// TIA Portal V16 export
// export: Created 2024-12-03T15:41:46.0079114Z, ExportSetting WithReadOnly, DisplayName Totally Integrated Automation Portal, DisplayVersion V16 Update 6, DisplayName TIA Portal Version Control Interface, DisplayVersion V16 Update 2, DisplayName TIA Portal Openness, DisplayVersion V16 Update 6, DisplayName TIA Portal Teamcenter Gateway, DisplayVersion V16, DisplayName SINAMICS Startdrive Advanced, DisplayVersion V16 Update 5, DisplayName SINAMICS Startdrive G130, G150, S120, S150, SINAMICS MV, S210, DisplayVersion V16 Update 5, DisplayName SINAMICS Startdrive G110M, G120, G120C, G120D, G120P, G115D, DisplayVersion V16 Update 5, DisplayName STEP 7 Professional, DisplayVersion V16 Update 6, DisplayName STEP 7 Safety, DisplayVersion V16, DisplayName WinCC Advanced / Unified PC, DisplayVersion V16 Update 6
TYPE "ConveyorTimes_UDT"
// stored: CreationDate 2021-07-13T07:41:36.2278727Z, InterfaceModifiedDate 2021-04-02T14:08:36.3341629Z, IsConsistent true, LibraryConformanceStatus The object is library-conformant., ModifiedDate 2021-07-03T12:49:45.956224Z
   STRUCT
      DelayedStart { S7_SetPoint := 'True'} : Time;
      ConveyorLength { S7_SetPoint := 'True'} : Real := 50000.0;
      InitDistance { S7_SetPoint := 'True'} : Real := 5000.0;
      ReceiveDistance { S7_SetPoint := 'True'} : Real := 0.0;   // TIme the ready to receive signal will stay on when conveyor is not empty
      SendDistance { S7_SetPoint := 'True'} : Real := 100.0;   // Time the ready to sent signal will stay on afther the end sensor turns false
      SleepDistance { S7_SetPoint := 'True'} : Real := 100000.0;
      GapDistance { S7_SetPoint := 'True'} : Real;   // The time when the conveyor can start its new sequence
      StartupDelay { S7_SetPoint := 'True'} : Time := t#25ms;
   END_STRUCT;
END_TYPE
